TYPE T_Ctrl_SIf_PTS_Out :
STRUCT
END_STRUCT
END_TYPE

(* stored: Version 1.1.0.1, ProductVersion 3.1.0.25
   DUT T_Ctrl_SIf_PTS_Out: Id {5dc8a1c3-ae78-4f0e-b7df-342fcfbaa401} *)
